// TIA Portal V18 export
TYPE "AI8xI_In"
   STRUCT
      Ch0 : Int;
      Ch1 : Int;
      Ch2 : Int;
      Ch3 : Int;
      Ch4 : Int;
      Ch5 : Int;
      Ch6 : Int;
      Ch7 : Int;
   END_STRUCT;
END_TYPE
